// TIA Portal V17 export
// export: Created 2023-02-14T02:49:35.791013Z, ExportSetting WithDefaults, DisplayName Totally Integrated Automation Portal, DisplayVersion V17, DisplayName TIA Portal Openness, DisplayVersion V17, DisplayName TIA Portal Teamcenter Gateway, DisplayVersion V17, DisplayName TIA Portal Version Control Interface, DisplayVersion V17, DisplayName SINAMICS Startdrive Advanced, DisplayVersion V17, DisplayName SINAMICS Startdrive G130, G150, S120, S150, SINAMICS MV, S210, DisplayVersion V17, DisplayName SINAMICS Startdrive G110M, G120, G120C, G120D, G120P, G115D, DisplayVersion V17, DisplayName STEP 7 Professional, DisplayVersion V17, DisplayName STEP 7 Safety, DisplayVersion V17, DisplayName WinCC Professional, DisplayVersion V17
DATA_BLOCK "IO Digital Preparation_DB"   // DB14
VERSION : 0.1
// stored: AutoNumber true, DBAccessibleFromOPCUA true, DBAccessibleFromWebserver true, InstanceOfName IO Digital Preparation, InstanceOfType FB
"IO Digital Preparation"
   // VAR_INPUT
   //    init : Bool;
   //    Reset : Bool;
   // END_VAR
   // VAR
   //    "FS-01.01" { S7_SetPoint := 'True'} : "Digital";
   //    "DRP-P02.01" { S7_SetPoint := 'True'} : "Digital";
   //    "DRP-P02.02" { S7_SetPoint := 'True'} : "Digital";
   //    "DRP-P03.01" { S7_SetPoint := 'True'} : "Digital";
   //    "DRP-P03.02" { S7_SetPoint := 'True'} : "Digital";
   //    "DRP-P04.01" { S7_SetPoint := 'True'} : "Digital";
   //    "DRP-P05.01" { S7_SetPoint := 'True'} : "Digital";
   //    "DRP-P05.02" { S7_SetPoint := 'True'} : "Digital";
   //    "DRP-P06.01" { S7_SetPoint := 'True'} : "Digital";
   //    "DRP-P07.01" { S7_SetPoint := 'True'} : "Digital";
   //    "DRP-P08.01" { S7_SetPoint := 'True'} : "Digital";
   //    "DRP-P09.01" { S7_SetPoint := 'True'} : "Digital";
   //    "DRP-P09.02" { S7_SetPoint := 'True'} : "Digital";
   //    "LL-51.01" { S7_SetPoint := 'True'} : "Digital";
   //    "ML-51.01" { S7_SetPoint := 'True'} : "Digital";
   //    "HL-51.01" { S7_SetPoint := 'True'} : "Digital";
   // END_VAR
BEGIN
END_DATA_BLOCK
